// TwinCAT 3 PLC project OvenProj
// ProgramVersion: 3.1.4023.0
// libraries:
//   Tc2_Standard, * (Beckhoff Automation GmbH)
//   Tc2_System, * (Beckhoff Automation GmbH)
//   Tc3_Module, * (Beckhoff Automation GmbH)
// project tree:
//   / GlobalTextList.TcGTLO, PlcTask.TcTTO, Visualization Manager.TcVMO (not stored)
//   POUs/ MAIN.TcPOU, Oven.TcPOU, Pizza.TcPOU
//   VISUs/ Visualization.TcVIS
// real-time tasks:
//   TASK PlcTask: cycle T#10ms, priority 20, ADS port 350

CONFIGURATION OvenProj
    RESOURCE PLC ON TwinCAT3
        TASK PlcTask(INTERVAL := T#10ms, PRIORITY := 20);
        PROGRAM MAIN WITH PlcTask : MAIN;
    END_RESOURCE
END_CONFIGURATION

// ---- POUs/MAIN.TcPOU
PROGRAM MAIN
VAR
	MyOven:oven;
	Step_Stat:INT:=0;
	MyPizza:Pizza;
END_VAR

//IF MyOven.Power THEN
//	CASE Step_Stat OF
//		0:
//		//MyOven.BlinkAlarm();
//		MyOven.MovePizzaToDeck();
//		IF MyOven.MovePizzaToOven() THEN
//			Step_Stat:=Step_Stat+1;
//		END_IF
//		1: 
//		MyOven.MovePizzaToDeck();
//		IF MyOven.BakeThePizza() THEN
//			Step_Stat:=Step_Stat+1;
//		END_IF
//		2:
//		MyOven.MovePizzaToDeck();
//		IF MyOven.MovePizzaOutTheOven() THEN
//			Step_Stat:=0;
//		ELSE
//			MyOven.OverBaked(); 
////				IF MyOven.Burned THEN
////					MyOven.BlinkAlarm();
////				END_IF	
//		END_IF
//		99:
//		IF MyOven.Init() THEN
//			Step_Stat:=0;
//		END_IF
//	END_CASE
//END_IF

if MyOven.Power then
	CASE Step_Stat OF
		0:
			MyOven.Init();
			Step_Stat:=Step_Stat+1;
		1:
			MyOven.MovePizzaToDeck();
			Step_Stat:=Step_Stat+1;
		2:
			MyOven.MovePizzaToOven();
			Step_Stat:=Step_Stat+1;
		3:
			 IF MyOven.BakeThePizza() THEN
				 MyOven.OverBaked();
				Step_Stat:=Step_Stat+1; 
				ELSE
					Step_Stat:=Step_Stat+1; 
			 END_IF
			
		4:
			IF MyOven.Alarm THEN
				MyOven.BlinkAlarm();
			END_IF
			MyOven.MovePizzaOutTheOven();
			Step_Stat:=1;
	
	END_CASE
END_IF

END_PROGRAM

// ---- POUs/Oven.TcPOU
FUNCTION_BLOCK Oven
VAR_INPUT
END_VAR
VAR_OUTPUT
END_VAR
VAR
	Power :BOOL;
	PizzaReady:BOOL;
	PizzaOndeck:BOOL;
	PizzaInOven :BOOL;
	PizzaDone:BOOL;
	PizzaIsBaked:BOOL;
	Burned:BOOL; 
	Alarm:BOOL;
	OvenTimer:TON;
	MoveTimer:TON;
	AlarmTimer:TON;
	OverBackedTimer:TON;
	OverCocked:TON;
	OffTimer:TON;
	Blink:INT:=0;
	AlarmCounter: int:=0;
END_VAR

METHOD BakeThePizza : BOOL
VAR_INPUT
END_VAR
IF PizzaInOven AND Power THEN
	OvenTimer(IN:=TRUE,PT:=T#5S);
	IF OvenTimer.Q THEN
		OverCocked(IN:=TRUE,PT:=T#5S);
		PizzaIsBaked:=TRUE;
		BakeThePizza:=TRUE;	
	END_IF
END_IF
END_METHOD

METHOD BlinkAlarm : BOOL
CASE Blink OF
	0:
	IF  AlarmCounter<4 THEN
		Alarm:=TRUE;
		AlarmCounter:=AlarmCounter+1;
		Blink:=Blink+1;
	ELSE
		Power:=FALSE;	
	END_IF

	1:
		AlarmTimer(IN:=TRUE,PT:=T#500MS);
		IF AlarmTimer.Q THEN
			AlarmTimer(IN:=FALSE);
			Blink:=Blink+1;
		END_IF
	
	2:
		Alarm:=FALSE;
		Blink:=Blink+1;
		
	3:
		OffTimer(IN:=TRUE,PT:=T#200MS);
		IF OffTimer.Q THEN
			OffTimer(IN:=FALSE);
			Blink:=0;
			AlarmCounter:=AlarmCounter+1;
		END_IF
		
END_CASE
END_METHOD

METHOD Init : BOOL
VAR_INPUT
END_VAR
	OvenTimer(IN:=FALSE);
	OverBackedTimer(IN:=FALSE);
	PizzaInOven:=FALSE;
	Burned:=FALSE;
	PizzaIsBaked:=FALSE;
	Init:=TRUE;
	Alarm:=FALSE;
	AlarmCounter:=0;
END_METHOD

METHOD MovePizzaOutTheOven : BOOL
VAR_INPUT
END_VAR
VAR
	et:Time;
END_VAR
IF PizzaInOven AND PizzaIsBaked AND NOT PizzaDone AND NOT Burned THEN 
	MoveTimer(in:=TRUE,PT:=T#500MS);
	et:=MoveTimer.ET;
	IF MoveTimer.Q THEN
		PizzaInOven:=FALSE;
		PizzaIsBaked:=FALSE;
		PizzaDone:=TRUE;
		OvenTimer(IN:=FALSE);
		MovePizzaOutTheOven:=TRUE;
//		IF Burned THEN
//			DoneBurned:=TRUE;
//		END_IF
		MoveTimer(IN:=FALSE);
	END_IF
END_IF
END_METHOD

METHOD MovePizzaToDeck : BOOL
VAR_INPUT
END_VAR
IF PizzaReady AND NOT PizzaOndeck THEN
MoveTimer(IN:=TRUE,PT:=T#500MS);
	IF MoveTimer.Q THEN
		PizzaReady:=FALSE;
		PizzaOndeck:=TRUE;
		MoveTimer(IN:=FALSE);
		MovePizzaToDeck:=TRUE;
	END_IF	
END_IF
END_METHOD

METHOD MovePizzaToOven : BOOL
VAR_INPUT
END_VAR
IF PizzaOndeck AND NOT PizzaInOven THEN
MoveTimer(IN:=TRUE,PT:=T#500MS);
	IF MoveTimer.Q THEN
		PizzaOndeck:=FALSE;
		PizzaInOven:=TRUE;
		MoveTimer(IN:=FALSE);
		MovePizzaToOven:=TRUE;
	END_IF	
END_IF
END_METHOD

METHOD OverBaked : BOOL
VAR_INPUT
END_VAR
IF PizzaDone AND PizzaInOven THEN
	OverBackedTimer(IN:=TRUE,PT:=T#3S);
	IF OverBackedTimer.Q THEN
		Burned:=TRUE;
		PizzaIsBaked:=FALSE;
		OverBackedTimer(IN:=FALSE);
		alarm:=TRUE;
		OverBaked:=TRUE;
	END_IF
END_IF
END_METHOD

END_FUNCTION_BLOCK

// ---- POUs/Pizza.TcPOU
FUNCTION_BLOCK Pizza
VAR
	Exists :BOOL;
	IsBacked:BOOL;
	BakingTime:Time;
END_VAR

END_FUNCTION_BLOCK

// ---- GlobalTextList.TcGTLO
TEXTLIST GlobalTextList
  815 = '%S'
  585 = '%s'
  501 = '%ss'
  816 = '%y'
  692 = "'Baker Stand"
  251 = 'as'
  545 = 'Baker Stand'
  495 = 'Belt Move Time: %s'
  902 = 'Belt Moving Time : %H:%M:%S'
  457 = 'Belt Moving Time : %H:%M:%s'
  216 = 'Belt Moving Time : %o'
  964 = 'Belt Moving Time : %S'
  94 = 'Belt Moving Time :%S'
  725 = 'Belt Moving Time :%s'
  595 = 'Belt Moving Time :%t %s'
  988 = 'Belt Moving Time :%t%s'
  437 = 'Moving Time : %s'
  901 = 'Moving Time : %S'
  774 = 'Moving Time : %X'
  180 = 'Pizza Ready'
  358 = 'Pizza Ready >>>'
  10 = 'Put away'
  739 = 'Send The Pizza'
  56 = 'Send The Pizza >>>'
  484 = 'STIPIZZA'
  958 = 'STIWA-PIZZA'
  472 = 'Time : %s'
  837 = 'Time : %S'
  936 = 'Trash Pin'
END_TEXTLIST

// ---- VISUs/Visualization.TcVIS
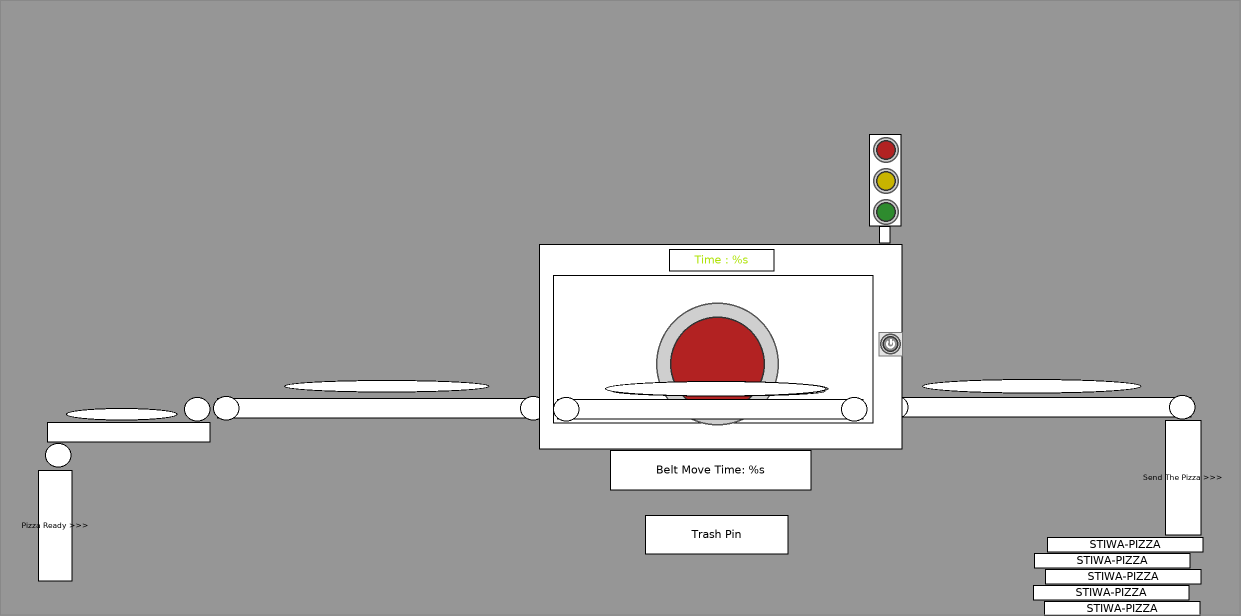
VISUALIZATION Visualization  // 1241x616
    RoundedRectangle (217,398 325x20)
    Ellipse (520,396 26x24)
    RoundedRectangle (866,397 325x20)
    Ellipse (1169,395 26x24)
    Ellipse (213,396 26x24)
    RoundedRectangle (47,422 163x20), angle 343
    Ellipse (45,443 26x24)
    Ellipse (184,397 26x24)
    Ellipse (66,408 111x12), angle 343, invisible if: NOT MAIN.MyOven.PizzaReady
    Ellipse (284,380 205x12), invisible if: NOT MAIN.MyOven.PizzaOndeck
    Ellipse (922,379 219x14), invisible if: NOT MAIN.MyOven.PizzaDone
    Rectangle (1126,459 115x36), angle 90, "Send The Pizza >>>"
        OnMouseClick: execute { MAIN.MyOven.PizzaDone:=FALSE; }
    Rectangle (0,509 111x34), angle 270, "Pizza Ready >>>"
        OnMouseClick: execute { MAIN.MyOven.PizzaReady:=TRUE; }
    Rectangle (610,450 201x40), "Belt Move Time: %s", text variable: Time_to_int(MAIN.MyOven.MoveTimer.ET)/1000
    Rectangle (1044,601 156x15), "STIWA-PIZZA"
    Rectangle (1033,585 156x15), "STIWA-PIZZA"
    Rectangle (1045,569 156x15), "STIWA-PIZZA"
    Rectangle (1034,553 156x15), "STIWA-PIZZA"
    Rectangle (1047,537 156x15), "STIWA-PIZZA"
    Rectangle (645,515 143x39), "Trash Pin"
        OnMouseClick: execute { MAIN.Step_Stat:=0; }
    Ellipse (882,395 26x24)
    Rectangle (539,244 363x205)
    RoundedRectangle (553,275 320x148)
    Lamp1 (646,279 143x170), variable: MAIN.MyOven.Power, style: Lamp-Lamp1-Red
    RoundedRectangle (557,399 306x20)
    Ellipse (841,397 26x24)
    Ellipse (553,397 26x24)
    PowerSwitch (877,332 27x24), variable: MAIN.MyOven.Power, behaviour: TOGGLE, style: Switch-PowerSwitch-Gray
    Rectangle (669,249 105x22), "Time : %s", text variable: Time_to_Int(MAIN.MyOven.OvenTimer.ET)/1000
    Ellipse (612,386 213x10), invisible if: NOT MAIN.MyOven.PizzaInOven
    Ellipse (607,381 221x15), invisible if: NOT MAIN.MyOven.PizzaIsBaked
    Ellipse (605,381 221x15), invisible if: NOT MAIN.MyOven.Burned
    RoundedRectangle (869,134 32x92)
    Lamp1 (871,197 30x30), variable: MAIN.MyOven.Power, style: Lamp-Lamp1-Green
    Lamp1 (871,135 30x30), variable: NOT MAIN.MyOven.Power, style: Lamp-Lamp1-Red
    Lamp1 (871,166 30x30), variable: MAIN.MyOven.Alarm, style: Lamp-Lamp1-Yellow
    Rectangle (879,226 11x17)
END_VISUALIZATION
